// Provide logging 
FUNCTION_BLOCK FB_TcAlarming IMPLEMENTS I_Logging
VAR_INPUT
	eLogLevel:				E_LogLevel:= E_LogLevel.Verbose;
END_VAR
VAR_OUTPUT
END_VAR
VAR
	iLogging:				I_Logging;
	aAlarm:					ARRAY[0..99] OF FB_TcAlarm; // Message store
    nAlarm:					UINT := 0;                     // Message count
END_VAR

// IF NOT bInit THEN
// 	bInit:= TRUE;
// 	aAlarm[0].
// 	aAlarm[0].CreateEx(TC_EVENTS.TcLogging.Verbose, FALSE, 0);
// END_IF
// 
// IF fbAlarm.bRaised THEN
// 	;
// ELSE
// 	fbAlarm.Raise(0);
// END_IF

METHOD PUBLIC M_Attach : BOOL
VAR_INPUT
	iLogging:				I_Logging;
END_VAR
IF THIS^.iLogging = 0 THEN
	THIS^.iLogging:= iLogging;
	M_Attach:= TRUE;
ELSIF THIS^.iLogging = iLogging THEN
	// already inside
	M_Attach:= TRUE;
	RETURN;
ELSE
	// redirect to next logging function block
	THIS^.iLogging.M_Attach(iLogging);
END_IF
END_METHOD

METHOD PUBLIC M_Log : BOOL
VAR_INPUT
	stMessage:			ST_Message;
END_VAR
VAR
	fbSourceInfo:		FB_TcSourceInfo;
END_VAR
// IF THIS^.eLogLevel > eLogLevel THEN
// 	M_Log:= TRUE;
// 	RETURN;
// END_IF
// 
// fbSourceInfo.Clear();
// fbSourceInfo.sName:= stMessage.sSource;
// 
// CASE eLogLevel OF
// 	E_LogLevel.Verbose:
//     	fbMsg.CreateEx(TC_EVENTS.TcLogging.Verbose, fbSourceInfo); 	
// 
// 	E_LogLevel.Info:
//     	fbMsg.CreateEx(TC_EVENTS.TcLogging.Info, fbSourceInfo); 
// 		
// 	E_LogLevel.Warning:		
//     	fbMsg.CreateEx(TC_EVENTS.TcLogging.Warning, fbSourceInfo); 
// 		
// 	E_LogLevel.Error:
//     	fbMsg.CreateEx(TC_EVENTS.TcLogging.Error, fbSourceInfo); 
// 		
// 	E_LogLevel.Critical:
//     	fbMsg.CreateEx(TC_EVENTS.TcLogging.Critical, fbSourceInfo); 
// 		
// END_CASE
// 
// fbMsg.ipArguments.Clear().AddString(stMessage.sDefault);
// 
// fbMsg.Send(stMessage.nTimestamp);
END_METHOD

PROPERTY PUBLIC P_LogLevel : E_LogLevel
GET
P_LogLevel:= eLogLevel;
END_GET
SET
eLogLevel:= P_LogLevel;
END_SET
END_PROPERTY

END_FUNCTION_BLOCK

(* stored: Version 1.1.0.1
   POU FB_TcAlarming: Id {b6b9d53e-320a-43f4-af08-5491e8ff7b78}, SpecialFunc None
   Method M_Attach: Id {a40614b1-3973-468c-ab07-88a8adebeba6}
   Method M_Log: Id {5a47f799-51ce-40a3-86ed-99adceead7ba}
   Property P_LogLevel: Id {dacde164-261f-416f-89f3-89fe3a30d375}
   Get Get: Id {2cc2483d-8888-40ac-a1a2-5c89fae1112b}
   Set Set: Id {53395058-5225-4b5a-bfa4-8537b852ef8e} *)
